INTERFACE I_EventHandlerItem EXTENDS I_Disposable

METHOD PUBLIC Emit : BOOL
VAR_INPUT
	EventName : T_MaxString;
	Event : I_Event;
END_VAR
END_METHOD

METHOD PUBLIC EqualTo : BOOL
VAR_INPUT
	Name : T_MaxString;
	Handler : I_EventHandler;
END_VAR
END_METHOD

PROPERTY PUBLIC Next : I_EventHandlerItem
GET
END_GET
SET
END_SET
END_PROPERTY

PROPERTY PUBLIC Previous : I_EventHandlerItem
GET
END_GET
SET
END_SET
END_PROPERTY

END_INTERFACE

(* stored: Version 1.1.0.1, ProductVersion 3.1.4026.13
   Itf I_EventHandlerItem: Id {943820f2-6d02-43f4-a224-eda85ce6c166}
   Method Emit: Id {d47a8275-0b77-488c-b526-2a215b45aa18}
   Method EqualTo: Id {1e507b2d-2942-4a96-9a80-d7fb383970fc}
   Property Next: Id {f5301b65-90eb-4f3e-be99-c549aec9e832}
   Get Get: Id {027001e4-6c4f-42c3-b1e5-087bb744cc00}
   Set Set: Id {3262ecdb-ae07-4100-970b-4d9860bea05f}
   Property Previous: Id {9796fcda-cc4f-4756-aab0-ff05fc1b2173}
   Get Get: Id {4a6f9eeb-51b6-4a64-88c4-3a3a67de0e8b}
   Set Set: Id {b6ceee62-4951-4759-89fd-f2405609e1a4} *)
